(* IEC 61131-3 sources: CS_4_Aufzugsteuerung/src/Stations/CP112/Steuerung/Class/clsMotorControl, 1 file *)

(* ---- clsMotorControl.st ---- *)
(*!
<Class
	Name               = "clsMotorControl"
	Revision           = "0.0"
	RealtimeTask       = "true"
	CyclicTask         = "false"
	DefCyclictime      = "1 ms"
	BackgroundTask     = "false"
	Sigmatek           = "false"
	OSInterface        = "false"
	HighPriority       = "false"
	Automatic          = "false"
	UpdateMode         = "Prescan"
	SharedCommandTable = "true"
	Objectsize         = "(480,600)">
	<Channels>
		<Server Name="ClassSvr" Visualized="false" Remotely="true" Initialize="false" WriteProtected="false" Retentive="false"/>
		<Server Name="sAcceleration" Visualized="false" Initialize="false" WriteProtected="false" Retentive="false"/>
		<Server Name="sCmd" Visualized="false" Initialize="false" WriteProtected="false" Retentive="false"/>
		<Server Name="sDistance" Visualized="false" Initialize="false" WriteProtected="false" Retentive="false"/>
		<Server Name="sMode" Visualized="false" Initialize="false" WriteProtected="true" Retentive="false"/>
		<Server Name="sPosition" Visualized="false" Initialize="false" WriteProtected="false" Retentive="false"/>
		<Server Name="sState" Visualized="false" Initialize="false" WriteProtected="true" Retentive="false"/>
		<Server Name="sVelocity" Visualized="false" Initialize="false" WriteProtected="false" Retentive="false"/>
		<Client Name="cAxis" Required="true" Internal="false"/>
	</Channels>
	<Separators>
		<Servers>
			<SepChn Name="TEST" Position="7"/>
		</Servers>
	</Separators>
</Class>
*)
clsMotorControl : CLASS
	TYPE
	  MOTOR_CMD :  //! <Type Public="true" Name="MOTOR_CMD"/>
	  (
	    MOVE_ABS,
	    MOVE_REL,
	    STOP,
	    POWER_ON,
	    POWER_OFF,
	    MOVE_INFINITE,
	    STOP_EMG
	  )$UDINT;
	  MOTOR_ERROR :
	  (
	    EnumItem0
	  )$UDINT;
	  MOTOR_MODE :  //! <Type Public="true" Name="MOTOR_MODE"/>
	  (
	    IDLE,
	    MOVE_ABS,
	    MOVE_REL,
	    POWER_ON,
	    POWER_OFF,
	    STOP,
	    STOP_EMG,
	    MOVE_INFINITE
	  )$UDINT;
	END_TYPE
  //Servers:
	ClassSvr 	: SvrChCmd_DINT;
	sMode 	: SvrCh_MOTOR_MODE_PTofCls_clsMotorControl;
	sState 	: SvrCh_DINT;
	sPosition 	: SvrCh_DINT;
	sDistance 	: SvrCh_DINT;
	sVelocity 	: SvrCh_DINT;
	sAcceleration 	: SvrCh_DINT;
	sCmd 	: SvrCh_MOTOR_CMD_PTofCls_clsMotorControl;
  //Clients:
	cAxis 	: CltChCmd__LMCAxis;
  //Variables:
  //Functions:

	FUNCTION VIRTUAL GLOBAL RtWork
		VAR_INPUT
			EAX 	: UDINT;
		END_VAR
		VAR_OUTPUT
			state (EAX) 	: UDINT;
		END_VAR;

	FUNCTION GLOBAL moveABS
		VAR_INPUT
			position 	: DINT;
			velocity 	: DINT;
			acceleration 	: DINT;
		END_VAR;

	FUNCTION GLOBAL moveREL
		VAR_INPUT
			distance 	: DINT;
			velocity 	: DINT;
			acceleration 	: DINT;
		END_VAR;

	FUNCTION GLOBAL moveInfinite
		VAR_INPUT
			velocity 	: DINT;
			acceleration 	: DINT;
		END_VAR;

	FUNCTION GLOBAL powerOn;

	FUNCTION GLOBAL powerOff;

	FUNCTION GLOBAL stopEMG;

	FUNCTION GLOBAL stopNORMAL;

	FUNCTION GLOBAL isReady
		VAR_OUTPUT
			isReady 	: DINT;
		END_VAR;

	FUNCTION VIRTUAL GLOBAL sCmd::Write
		VAR_INPUT
			input (EAX) 	: clsMotorControl::MOTOR_CMD;
		END_VAR
		VAR_OUTPUT
			result (EAX) 	: clsMotorControl::MOTOR_CMD;
		END_VAR;
  //Tables:
	FUNCTION @STD
		VAR_OUTPUT
			ret_code	: CONFSTATES;
		END_VAR;
	FUNCTION GLOBAL TAB @CT_;
END_CLASS;

#pragma usingLtd _LMCAxis

FUNCTION VIRTUAL GLOBAL clsMotorControl::sCmd::Write
	VAR_INPUT
		input (EAX) 	: clsMotorControl::MOTOR_CMD;
	END_VAR
	VAR_OUTPUT
		result (EAX) 	: clsMotorControl::MOTOR_CMD;
	END_VAR

	sCmd := input;

  IF sCmd = MOTOR_CMD::POWER_ON THEN
    powerOn();
  END_IF;

  IF sCmd = MOTOR_CMD::POWER_OFF THEN
    powerOff();
  END_IF;

  IF sCmd = MOTOR_CMD::MOVE_ABS THEN
    moveAbs(sPosition,sVelocity, sAcceleration);
  END_IF;

  IF sCmd = MOTOR_CMD::MOVE_REL THEN
    moveREL(distance:=sDistance, velocity:=sVelocity, acceleration:=sAcceleration);
  END_IF;

  IF sCmd = MOTOR_CMD::MOVE_INFINITE THEN
    moveInfinite(velocity:=sVelocity, acceleration:=sAcceleration);
  END_IF;

  IF sCmd = MOTOR_CMD::STOP THEN
    stopNORMAL();
  END_IF;

  IF sCmd = MOTOR_CMD::STOP_EMG THEN
    stopEMG();
  END_IF;

	result := sCmd;

END_FUNCTION

FUNCTION GLOBAL clsMotorControl::moveABS
	VAR_INPUT
		position 	: DINT;
		velocity 	: DINT;
		acceleration 	: DINT;
	END_VAR

  sPosition := position;
  sVelocity := velocity;
  sAcceleration := acceleration;

  sState := 1;
  sMode := MOTOR_MODE::MOVE_ABS;
END_FUNCTION

FUNCTION GLOBAL clsMotorControl::powerOn
   sState := 1;
   sMode := MOTOR_MODE::POWER_ON;
END_FUNCTION

FUNCTION GLOBAL clsMotorControl::powerOff
  sState := 1;
  sMode := MOTOR_MODE::POWER_OFF;
END_FUNCTION

FUNCTION GLOBAL clsMotorControl::stopNORMAL
  sState := 1;
  sMode := MOTOR_MODE::STOP;
END_FUNCTION

FUNCTION GLOBAL clsMotorControl::stopEMG
  sState := 1;
  sMode := MOTOR_MODE::STOP_EMG;
END_FUNCTION

FUNCTION GLOBAL clsMotorControl::moveREL
	VAR_INPUT
		distance 	: DINT;
		velocity 	: DINT;
		acceleration 	: DINT;
	END_VAR

  sDistance := distance;
  sVelocity := velocity;
  sAcceleration := acceleration;

  sState := 1;
  sMode := MOTOR_MODE::MOVE_REL;

 END_FUNCTION

FUNCTION GLOBAL clsMotorControl::moveInfinite
	VAR_INPUT
		velocity 	: DINT;
		acceleration 	: DINT;
	END_VAR

  sVelocity := velocity;
  sAcceleration := acceleration;

  sState := 1;
  sMode := MOTOR_MODE::MOVE_INFINITE;
END_FUNCTION

FUNCTION GLOBAL clsMotorControl::isReady
	VAR_OUTPUT
		isReady 	: DINT;
	END_VAR

  IF cAxis.AxisStatus.PowerOn AND cAxis.AxisStatus.Standstill AND cAxis.AxisError <> 0 THEN
    isReady := TRUE;
    RETURN;
  end_if;

  isReady := FALSE;

END_FUNCTION

FUNCTION VIRTUAL GLOBAL clsMotorControl::RtWork
	VAR_INPUT
		EAX 	: UDINT;
	END_VAR
	VAR_OUTPUT
		state (EAX) 	: UDINT;
	END_VAR

  CASE sMode OF

    MOTOR_MODE::IDLE:;

    MOTOR_MODE::STOP:
        cAxis.StopMove(Decel:=600000, Jerk:=1);
        sState := 0;
        sMode := MOTOR_MODE::IDLE;

    MOTOR_MODE::STOP_EMG:
        cAxis.QuickStop(Decel:=999999999);
        sState := 0;
        sMode := MOTOR_MODE::IDLE;

    MOTOR_MODE::POWER_ON:
        CASE sState OF

          1: IF cAxis.AxisStatus.ReadyToPowerOn THEN
              cAxis.PowerOn(Mode:= ::_LMCAXIS_MOVEDIRECTION::LMCAXIS_MOVE_ANY_WAY);
              sState := 2;
             END_IF;

          2: IF cAxis.AxisStatus.PowerOn THEN
              sState := 0;
              sMode := MOTOR_MODE::IDLE;
             END_IF;

        END_CASE;

     MOTOR_MODE::POWER_OFF:
        cAxis.PowerOff(Mode:=::_LMCAXIS_POWER_OFF_MODE::LMCAXIS_SMOOTH_STOPP);
        sState := 0;
        sMode := MOTOR_MODE::IDLE;

     MOTOR_MODE::MOVE_ABS:
        CASE sState OF

          1: IF cAxis.AxisStatus.PowerOn THEN
              cAxis.MoveAbsolute(Position:=sPosition, Speed:=sVelocity, Accel:=sAcceleration, Decel:=sAcceleration, Jerk:=1);
              sState := 2;
             END_IF;

          2: IF cAxis.AxisStatus.InPosition THEN
              sState := 0;
              sMode := MOTOR_MODE::IDLE;
             END_IF;

        END_CASE;

      MOTOR_MODE::MOVE_REL:
        CASE sState OF

          1: IF cAxis.AxisStatus.PowerOn THEN
                cAxis.MoveRelative(Position:=sDistance, Mode:= _LMCAXIS_MOVE_RELATIVE_MODE::LMCAXIS_MOVE_RELATIVE_TO_DESTINATION, Speed:=sVelocity, Accel:=sAcceleration, Decel:=sAcceleration, Jerk:=1);
              sState := 2;
             END_IF;

          2: IF cAxis.AxisStatus.InPosition THEN
              sState := 0;
              sMode := MOTOR_MODE::IDLE;
             END_IF;

        END_CASE;

  END_CASE;

	state := READY;

END_FUNCTION
